(* CODESYS project EX4.project

Project tree, tasks and I/O mapping:
  Device : CODESYS Control Win V3, 3S - Smart Software Solutions GmbH, order no. 305021, version 3.5.11.30
    application Application
      libraries: Standard, * (System)
      task MainTask (cyclic, interval t#20ms, priority 1) calls PLC_PRG
      program PLC_PRG [LD]
*)

// Device/Application/PLC_PRG
PROGRAM PLC_PRG
VAR
   SB3 : BOOL;              // liga partida direta
   SB2 : BOOL;              // liga partida inversa
   SB1 : BOOL;              // para o motor
   H3 : BOOL;               //  Motor Ligado Partida Direta
   H2 : BOOL;               //  Motor Ligado Partida Inversa
   H1 : BOOL;               // Motor parado
   KM1 : BOOL;              // Partida direta
   KM2 : BOOL;              // Partida Inversa
   FR : BOOL;               // Sensor de Proteção de Falha
	AUX: BOOL;              // AUXILIAR
	STOP: BOOL;             // EMERGENCIA
	BREAK: BOOL;            // PARA TUDO
END_VAR

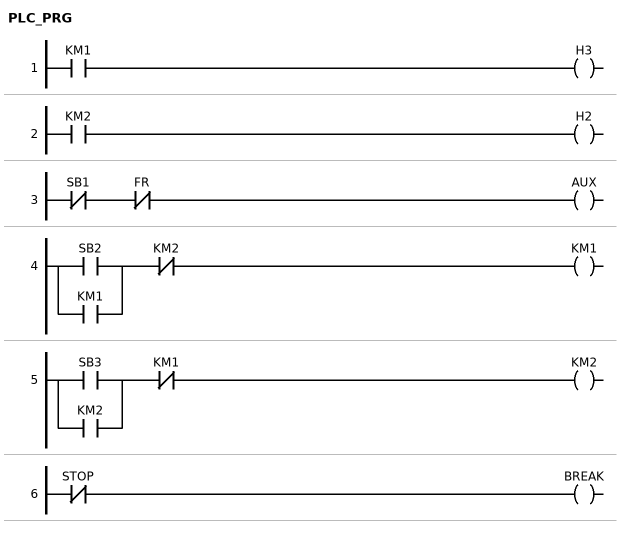
// NETWORK 1
H3 := KM1;

// NETWORK 2
H2 := KM2;

// NETWORK 3
AUX := NOT SB1 AND NOT FR;

// NETWORK 4
KM1 := (SB2 OR KM1) AND NOT KM2;

// NETWORK 5
KM2 := (SB3 OR KM2) AND NOT KM1;

// NETWORK 6
BREAK := NOT STOP;

END_PROGRAM
